FUNCTION FC_SQL_UpdateCommands : STRING(255)
VAR_INPUT
	iValue		:INT;
	iTag		:STRING;
END_VAR
VAR
END_VAR

FC_SQL_UpdateCommands:='UPDATE tags SET tagvalue = ';
FC_SQL_UpdateCommands:=CONCAT(STR1:=FC_SQL_UpdateCommands,STR2:=INT_TO_STRING(iValue));
FC_SQL_UpdateCommands:=CONCAT(STR1:=FC_SQL_UpdateCommands,STR2:=' ');
FC_SQL_UpdateCommands:=CONCAT(STR1:=FC_SQL_UpdateCommands,STR2:='WHERE tagname =  ');
FC_SQL_UpdateCommands:=CONCAT(STR1:=FC_SQL_UpdateCommands,STR2:=iTag);

END_FUNCTION

(* stored: Version 1.1.0.1, ProductVersion 3.1.4024.11
   POU FC_SQL_UpdateCommands: Id {fd6c82db-6dc4-4367-bf49-1658d2dd946a}, SpecialFunc None *)
